PROGRAM MAIN
VAR
END_VAR

PRG_PI_Regulator_ProgramExample();

END_PROGRAM

(* stored: Version 1.1.0.1, ProductVersion 3.1.4024.15
   POU MAIN: Id {10443e77-d6c6-4f80-af1f-4c159de3826a}, SpecialFunc None *)
